// TIA Portal V17 export
// export: Created 2023-12-22T15:02:59.4569135Z, ExportSetting WithDefaults, DisplayName Totally Integrated Automation Portal, DisplayVersion V17, DisplayName TIA Portal Openness, DisplayVersion V17, DisplayName TIA Portal Version Control Interface, DisplayVersion V17, DisplayName STEP 7 Professional, DisplayVersion V17, DisplayName STEP 7 Safety, DisplayVersion V17, DisplayName WinCC Advanced, DisplayVersion V17
ORGANIZATION_BLOCK "Cyclic interrupt"   // OB30, LAD, CyclicInterrupt
{ S7_Optimized_Access := 'TRUE' }
VERSION : 0.1
// stored: AutoNumber true, IsIECCheckEnabled false, SetENOAutomatically false
   VAR_INPUT
      Initial_Call : Bool;   // Initial call of this OB
      Event_Count : Int;   // Events discarded
   END_VAR
BEGIN

REGION Network 1
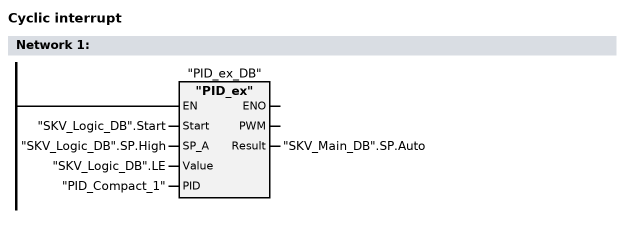
   RUNG wire#powerrail
      "PID_ex_DB"(Start := "SKV_Logic_DB".Start, SP_A := "SKV_Logic_DB".SP.High, Value := "SKV_Logic_DB".LE, PID := "PID_Compact_1", PWM =>, Result => "SKV_Main_DB".SP.Auto)
   END_RUNG
   // the same network as SCL:
   "PID_ex_DB"(Start := "SKV_Logic_DB".Start,   // "PID_ex"
               SP_A := "SKV_Logic_DB".SP.High,
               Value := "SKV_Logic_DB".LE,
               PID := "PID_Compact_1",
               Result => "SKV_Main_DB".SP.Auto);
END_REGION
END_ORGANIZATION_BLOCK
